PROGRAM MAIN
VAR
END_VAR

END_PROGRAM

(* stored: Version 1.1.0.1
   POU MAIN: Id {48a360ae-53c6-4935-a054-6aaa9b81a41d} *)
